// TIA Portal V17 export
// export: Created 2022-07-20T06:59:39.3129683Z, ExportSetting WithDefaults, DisplayName Totally Integrated Automation Portal, DisplayVersion V17, DisplayName TIA Portal Openness, DisplayVersion V17, DisplayName TIA Portal Version Control Interface, DisplayVersion V17, DisplayName SINAMICS Startdrive Advanced, DisplayVersion V17, DisplayName SINAMICS Startdrive G130, G150, S120, S150, SINAMICS MV, S210, DisplayVersion V17, DisplayName SINAMICS Startdrive G110M, G120, G120C, G120D, G120P, G115D, DisplayVersion V17, DisplayName STEP 7 Professional, DisplayVersion V17, DisplayName STEP 7 Safety, DisplayVersion V17, DisplayName WinCC Advanced, DisplayVersion V17
FUNCTION "FC10013_2IntToReal" : Void   // FC10013, LAD
TITLE = FC10013_2IntToReal
{ S7_Optimized_Access := 'TRUE' }
AUTHOR : Anirouddh
FAMILY : 1001x_CONVERT
VERSION : 1.0
// Release note : 
// 1.0 - Feature developped
// stored: AutoNumber false, IsIECCheckEnabled false, SetENOAutomatically false, UDAEnableTagReadback false
   VAR_INPUT
      HighWeight_Int : Int;
      LowWeight_Int : Int;
   END_VAR
   VAR_OUTPUT
      Output_Real : Real;
   END_VAR
   VAR_TEMP
      Temp1 : DWord;
      Temp2 : DWord;
   END_VAR
BEGIN

REGION Network 1 (SCL): 2 Ints To Real conversion
   #Temp1 := INT_TO_DWORD(#HighWeight_Int);
   #Temp2 := INT_TO_DWORD(#LowWeight_Int);

   #Temp1 := SHL_DWORD(IN := #Temp1, N := 16);

   #Temp1 := #Temp1 OR #Temp2;

   #Output_Real := DWORD_TO_REAL(#Temp1);
END_REGION
END_FUNCTION
